FUNCTION_BLOCK FB_CONCAT (* Concatenation of WSTRING inputs *)
  (* Standard: 61499-1 *)
  (* Version 0.0, 2001-04-12, JHC, Rockwell Automation, First XML version. *)
  (* Compiler header: package fb.rt.diag; *)
  (* Compiler Java IBM VisualAge 3.0 *)
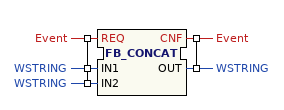
  EVENT_INPUT
    REQ WITH IN1, IN2;
  END_EVENT
  EVENT_OUTPUT
    CNF WITH OUT;
  END_EVENT
  VAR_INPUT
    IN1 : WSTRING;
    IN2 : WSTRING;
  END_VAR
  VAR_OUTPUT
    OUT : WSTRING;
  END_VAR
  ALGORITHM REQ IN JAVA:
public void service_REQ(boolean qi){
OUT.value=IN1.value+IN2.value;
CNF.serviceEvent(this);}
  END_ALGORITHM
END_FUNCTION_BLOCK
